{attribute 'pack_mode' := '1'}
    {attribute 'OPC.UA.DA' := '1'}
    {attribute 'OPC.UA.DA.StructuredType' := '1'}
    (*
    ST_RW_RealMb_HMI_IgnitionExp
    ==================================================
    Generated from Ignition UDT: RW_Real_MB
    Total tags: 1
    Generated on: 2025-09-15 12:47:19
    *)
    TYPE ST_RW_RealMb_HMI_IgnitionExp :
    STRUCT
        {attribute 'OPC.UA.DA' := '1'}
        {attribute 'OPC.UA.DA.Description' := '{Description}'}
        // {Description}
        Value : REAL := 0.0;
    END_STRUCT
    END_TYPE

(* stored: Version 1.1.0.1
   DUT ST_RW_RealMb_HMI_IgnitionExp: Id {2580dcf1-9c8e-49e2-b7e4-fad6513ad07b} *)
